FUNCTION F_ComputeStringSize : UDINT
VAR_INPUT
    anyString   : ANY_STRING;
END_VAR
VAR 
    nStrLen : UDINT;
END_VAR


nStrLen := LEN2(pString:= anyString.pValue);
F_ComputeStringSize := F_ComputeLengthSize(nStrLen) + nStrLen;

END_FUNCTION

(* stored: Version 1.1.0.1
   POU F_ComputeStringSize: Id {4c350631-d3e5-4511-87db-1c3d68f24411}, SpecialFunc None *)
